RoboDK station: ConveyorAndArm_ASSEMBLY.rdk

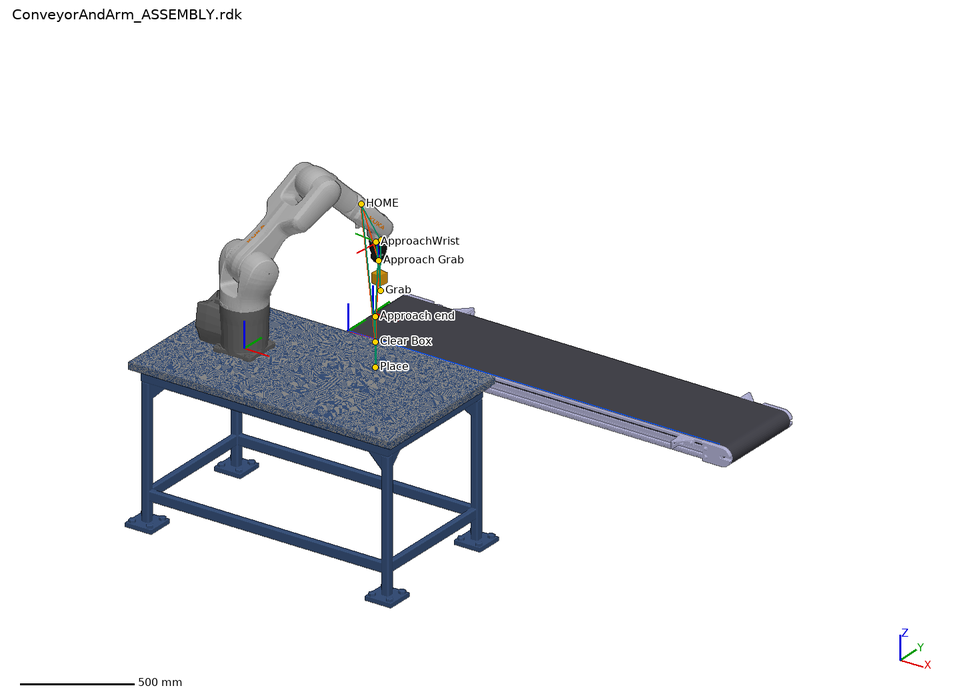
[picture v0: the station drawn from its stored meshes, robots at their saved joint values, targets as dots, program paths as lines]
Station ConveyorAndArm_ASSEMBLY (saved by RoboDK 5.5.0). Poses are relative to the parent item; angles as X-Y-Z fixed-axis rotations.
  - frame KUKA KR 6 R900-2 Base at (0, 0, 0) mm
    - robot KUKA KR 6 R900-2: 6 axes, payload 6.5 kg, reach 901 mm, repeatability 0.02 mm, weight 55 kg
        modified DH rows (alpha deg, a mm, theta deg, d mm): 0, 0, 0, 400; -90, 25, 0, 0; 0, 455, -90, 0; -90, 25, 0, 420; 90, 0, 0, 0; -90, 0, 180, 90
        joint limits [-170, -190, -120, -185, -120, -350] to [170, 45, 156, 185, 120, 350]; home [0, -90, 90, 0, 0, 0]; saved at [-66.498, -42.077, 85.836, 0.451, 44.725, 15.565]
      - frame RobotiQ 2F-85 Gripper (Mechanism) Base at (0, 0, 0) mm
        - robot RobotiQ 2F-85 Gripper (Mechanism) (model RobotiQ 2F85): 1 axes, payload 5 kg
            joint limits [0] to [85]; home [85]; saved at [49.9]
        - target OPEN (joint target) at (0, 0, 193.92) mm; joints [85] of RobotiQ 2F-85 Gripper (Mechanism)
        - target CLOSE (joint target) at (0, 0, 193.92) mm; joints [49.9] of RobotiQ 2F-85 Gripper (Mechanism)
      - tool Tool 1, TCP at (0, 0, 90) mm
        - object Cube 50mm at (-26.23, 21.37, 106.94) mm, rotated rx 179.99 ry 0.49 rz 3.34 deg, size 50 x 50 x 50 mm, geometry from Cube-50mm.sld
    - target HOME (Cartesian target) at (625, 0, 880) mm, rotated rx 0 ry 90 rz 0 deg; joints [0, -90, 90, 0, 0, 0] of KUKA KR 6 R900-2
    - target Approach Grab (Cartesian target) at (275.33, 630.64, 252.55) mm, rotated rx 178.96 ry 1.15 rz -167.25 deg; joints [-66.498, -42.077, 85.836, 0.451, 44.725, -54.054] of KUKA KR 6 R900-2
      - target ApproachWrist (Cartesian target) at (275.33, 630.64, 252.55) mm, rotated rx -178.91 ry -1.1 rz 9.78 deg; joints [-66.498, -42.077, 85.836, 0.451, 44.725, -54.054] of KUKA KR 6 R900-2
    - target Grab (Cartesian target) at (280.43, 639.86, 105.73) mm, rotated rx -179.96 ry 0.49 rz 4.75 deg; joints [-66.217, -27.279, 80.792, -0.758, 36.689, 119.143] of KUKA KR 6 R900-2
    - target Lift (Cartesian target) at (282.55, 639.87, 350.72) mm, rotated rx -179.96 ry 0.49 rz 4.75 deg; joints [-66.059, -47.483, 79.996, -0.535, 57.69, 118.98] of KUKA KR 6 R900-2
    - target Approach end (Cartesian target) at (699.44, 1.43, 350.65) mm, rotated rx 179.54 ry -0.21 rz 179.71 deg; joints [0, -47.48, 80, -0.54, 57.69, 0] of KUKA KR 6 R900-2
    - target Place (Cartesian target) at (698.54, 3.4, 103.62) mm, rotated rx 179.54 ry -0.21 rz 179.71 deg; joints [-0.161, -27.073, 80.727, -0.767, 36.556, 0.166] of KUKA KR 6 R900-2
    - target Clear Box (Cartesian target) at (698.98, 2.43, 225.66) mm, rotated rx 179.54 ry -0.21 rz 179.71 deg; joints [-0.082, -38.27, 82.701, -0.637, 45.779, 0.074] of KUKA KR 6 R900-2
  - object Table 1400x800x800mm at (0, 0, 0) mm, size 1420 x 820 x 800 mm, geometry from Table-1400x800x800mm.sld
  - frame Conveyor Belt (2m) Base at (271.92, 406.41, 0) mm, rotated rx 0 ry 0 rz 0.05 deg
    - robot Conveyor Belt (2m): 1 axes
        modified DH rows (alpha deg, a mm, theta deg, d mm): 0, 0, 0, 0 linear
        base shift (0, 0, 0) mm, rotated rx 0 ry 90 rz 0 deg
        joint limits [-10] to [2000]; home [0]; saved at [0]
      - frame Conveyor Object at (-16.59, 210, -1) mm, rotated rx 0 ry 0 rz 1.36 deg
    - target Pos_2 (joint target) at (0, 0, 0) mm; joints [0] of Conveyor Belt (2m)
    - target Pos_1 (joint target) at (1980.1, 0, 0) mm; joints [1980.1] of Conveyor Belt (2m)
  - program Conveyor Belt (3 instructions, listed below)
  - program ARM Take (17 instructions, listed below)
  - program ARM replace (17 instructions, listed below)
  - program H_OPEN (3 instructions, listed below)
  - program H_CLOSE (2 instructions, listed below)
  - program MAIN (10 instructions, listed below)
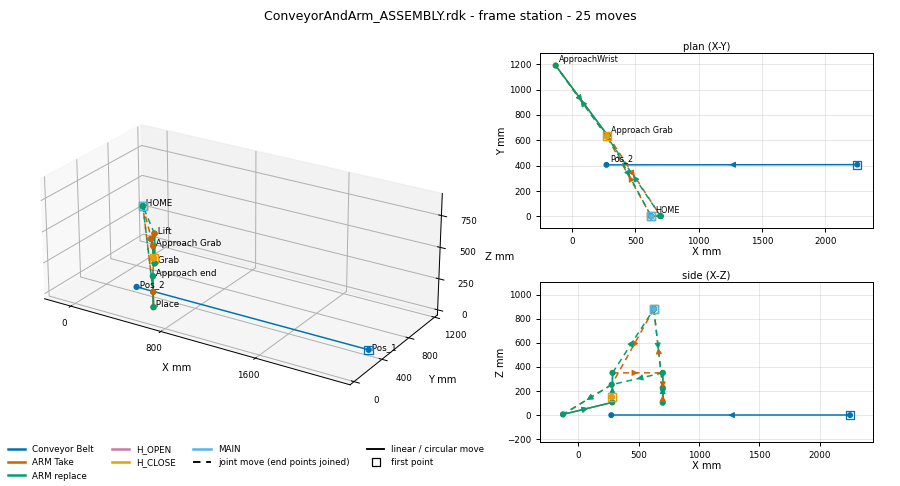
[picture p0: tool path of ConveyorAndArm_ASSEMBLY.rdk in frame station, 25 of 25 moves have a stored position in this frame; points joined in program order, loops and branches not executed]

--- program Conveyor Belt (robot Conveyor Belt (2m)) ---
  Set Ref.: Conveyor Belt (2m) Base
  MoveL (Pos_1)
  MoveL (Pos_2)

--- program ARM Take (robot KUKA KR 6 R900-2) ---
  Set Ref.: KUKA KR 6 R900-2 Base
  Set Tool: Tool 1
  MoveJ (HOME)
  MoveJ (Approach Grab)
  MoveJ (ApproachWrist)
  MoveL (Grab)
  Attach to Tool 1
  Call H_CLOSE
  Pause 500 ms
  MoveL (Lift)
  MoveJ (Approach end)
  MoveL (Place)
  Detach from Tool 1
  Call H_OPEN
  Pause 500 ms
  MoveL (Clear Box)
  MoveJ (HOME)

--- program ARM replace (robot KUKA KR 6 R900-2) ---
  Set Ref.: KUKA KR 6 R900-2 Base
  Set Tool: Tool 1
  MoveJ (HOME)
  MoveJ (Clear Box)
  MoveL (Place)
  Attach to Tool 1
  Call H_CLOSE
  Pause 500 ms
  MoveL (Approach end)
  MoveJ (Approach Grab)
  MoveJ (ApproachWrist)
  MoveL (Grab)
  Detach from Tool 1
  Call H_OPEN
  Pause 500 ms
  MoveL (Lift)
  MoveJ (HOME)

--- program H_OPEN (robot RobotiQ 2F-85 Gripper (Mechanism)) ---
  Set Ref.: RobotiQ 2F-85 Gripper (Mechanism) Base
  MoveJ (CLOSE)
  MoveJ (OPEN)

--- program H_CLOSE (robot RobotiQ 2F-85 Gripper (Mechanism)) ---
  MoveJ (OPEN)
  MoveJ (CLOSE)

--- program MAIN (robot KUKA KR 6 R900-2) ---
  Set Ref.: KUKA KR 6 R900-2 Base
  Set Tool: Tool 1
  Set speed (100.0 mm/s)
  MoveJ (HOME)
  Call Conveyor Belt
  Pause 500 ms
  Call ARM Take
  Pause 500 ms
  Call ARM replace
  Pause 500 ms
